// TIA Portal V20 export
TYPE "LER_typeRFIDInterface"
// stored: Access Published
   STRUCT
      commands : "LER_typeRFIDCommands";
      monitoring : "LER_typeRFIDMonitoring";
      configuration : "LER_typeRFIDConfiguration";
   END_STRUCT;
END_TYPE
